FUNCTION_BLOCK CTRL_PI_AR (* AR-Adapter-Wrapper um OSCAT CTRL_PI - bruckt zwischen adapter und OSCAT PI-Regler. Istwert, Sollwert, Hand-Umschaltung, Handwert, Reglerparameter UND Rauschunterdrueckung/Offset/Grenzwerte vollstaendig als Adapter-Sockets - kein explizites REQ mehr noetig. *)
  (* Standard: 61499-2; Description: Copyright (c) 2026 Meisterschulen am Ostbahnhof This program and the accompanying materials are made available under the terms of the Eclipse Public License 2.0 which is available at https://www.eclipse.org/legal/epl-2.0/ SPDX-License-Identifier: EPL-2.0 *)
  (* Version 1.3, 2026-10-03, Franz Höpfinger, Meisterschulen am Ostbahnhof, Franz: 'auch umstellen auf Adapter Only' (analog CTRL_PID_AR v1.3/1.4) - SUP/OFS/LL/LH von InputVars (REAL, With-gebunden an REQ) auf AR-Adapter-Sockets umgestellt (gleiches Muster wie KP/KI/M_I: *.E1 loest CTRL_PI.REQ aus, *.D1 liefert den Wert). Explizites REQ-EventInput (inkl. With-Bindungen) und CNF-EventOutput komplett entfernt - CTRL_PI.CNF->E_D_FF_ANY.CLK bleibt intern bestehen (fuer das Latch von Y/DIFF/LIM), nur der externe CNF-Durchgriff entfaellt. RST unveraendert. Sockets/Connections/Dokumentation zugleich auf die Reihenfolge der CTRL_PI-InputVars sortiert: AR_ACT, SET, SUP, OFS, M_I, AX_MAN, KP, KI, LL, LH. *)
  (* Version 1.2, 2026-09-19, Franz Höpfinger, Meisterschulen am Ostbahnhof, Bugfix: REQ hatte keine With-Verknuepfung zu SUP/OFS/LL/LH (IEC 61499 - ungebundene Vars werden nicht zuverlaessig gelesen), jetzt ergaenzt, gespiegelt vom inneren CTRL_PI. M_I/KP/KI von InputVars auf AR-Adapter-Sockets umgestellt (Konsistenz mit AR_ACT/SET). *)
  (* Version 1.1, 2026-09-15, Franz Höpfinger, Meisterschulen am Ostbahnhof, INIT/INITO entfernt (CTRL_PI kennt kein INIT, nur REQ/RST) - stattdessen echtes REQ-EventInput/CNF-EventOutput ergaenzt, direkt auf CTRL_PI.REQ/CNF gemappt. SET von InputVar auf AR-Socket umgestellt (dynamisch berechneter Sollwert, wie AR_ACT) - SET.E1 triggert CTRL_PI.REQ zusaetzlich zu AR_ACT.E1/AX_MAN.E1. *)
  (* Version 1.0, 2026-09-12, Franz Höpfinger, Meisterschulen am Ostbahnhof, Initial implementation of CTRL_PI_AR wrapper FB *)
  PACKAGE OSCAT_adapter::Control;
  (* Documentation:
  CTRL_PI_AR
   🇩🇪 Deutsch
   AR-Adapter-Wrapper um OSCAT::Basic::POUs::Engineering::Control::CTRL_PI. Istwert (AR_ACT), Sollwert (SET), Rauschunterdrueckung/Offset (SUP/OFS), Handwert (M_I), Handbetrieb-Umschaltung (AX_MAN), Reglerparameter (KP/KI) UND Grenzwerte (LL/LH) sind als Adapter-Sockets ausgefuehrt, in derselben Reihenfolge wie die InputVars des umschlossenen CTRL_PI - jeder loest bei Ankunft eines neuen Werts CTRL_PI.REQ aus. Kein explizites REQ-Event mehr noetig, da jeder Socket selbst triggert. RST (Reset des Integrators) bleibt als eigenes Event erhalten.
   Reine Adapter-Grenze
    - AR_ACT (Socket, AR): Istwert (REAL, z. B. von FT_DERIV_10_AR.AR_OUT)
   - SET (Socket, AR): Sollwert (REAL, dynamisch berechnet, z. B. Fahrgeschwindigkeit*Voreilung)
   - SUP (Socket, AR): Rauschunterdrueckung (REAL, dynamisch)
   - OFS (Socket, AR): Offset (REAL, dynamisch)
   - M_I (Socket, AR): Handwert (REAL, dynamisch)
   - AX_MAN (Socket, AX): Handbetrieb-Umschaltung (optional, z. B. von AX_T_FF.Q)
   - KP/KI (Socket, AR): Reglerparameter (REAL, dynamisch)
   - LL/LH (Socket, AR): unterer/oberer Grenzwert (REAL, dynamisch)
   - AR_Y (Plug, AR): Stellwert (REAL, z. B. zur Weitergabe an AR_TO_AD_NUM.AR_IN)
   - AR_DIFF (Plug, AR): Regelabweichung (DIFF = SET - ACT, REAL)
   - AB_LIM (Plug, AB): Begrenzung aktiv Flag (LIM, BOOL)
    🇬🇧 English
   AR-adapter wrapper around OSCAT::Basic::POUs::Engineering::Control::CTRL_PI. Actual value (AR_ACT), set point (SET), noise suppression/offset (SUP/OFS), manual value (M_I), manual mode switch (AX_MAN), controller gains (KP/KI) AND limits (LL/LH) are all adapter sockets, in the same order as the wrapped CTRL_PI's own InputVars, each triggering CTRL_PI.REQ on arrival - no explicit REQ event needed any more, since every socket triggers itself. RST (integrator reset) remains its own event. Control output (AR_Y), control error (AR_DIFF) and limit flag (AB_LIM) are adapter plugs.
  *)
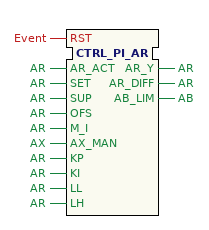
  EVENT_INPUT
    RST; (* Reset des Integrators (durchgereicht an CTRL_PI.RST) *)
  END_EVENT
  SOCKETS
    AR_ACT : adapter::types::unidirectional::AR; (* Istwert (REAL) *)
    SET : adapter::types::unidirectional::AR; (* Sollwert (REAL, dynamisch berechnet) *)
    SUP : adapter::types::unidirectional::AR; (* Rauschunterdrueckung (REAL, dynamisch) *)
    OFS : adapter::types::unidirectional::AR; (* Offset (REAL, dynamisch) *)
    M_I : adapter::types::unidirectional::AR; (* Handwert (REAL, dynamisch) *)
    AX_MAN : adapter::types::unidirectional::AX; (* Handbetrieb Umschaltung (BOOL/Event, optional) *)
    KP : adapter::types::unidirectional::AR; (* Proportionalbeiwert (REAL, dynamisch) *)
    KI : adapter::types::unidirectional::AR; (* Integralbeiwert (REAL, dynamisch) *)
    LL : adapter::types::unidirectional::AR; (* Unterer Grenzwert (REAL, dynamisch) *)
    LH : adapter::types::unidirectional::AR; (* Oberer Grenzwert (REAL, dynamisch) *)
  END_SOCKETS
  PLUGS
    AR_Y : adapter::types::unidirectional::AR; (* Stellwert (REAL) *)
    AR_DIFF : adapter::types::unidirectional::AR; (* Regelabweichung / Differenz (REAL) *)
    AB_LIM : adapter::types::unidirectional::AB; (* Begrenzung aktiv Flag (BOOL) *)
  END_PLUGS
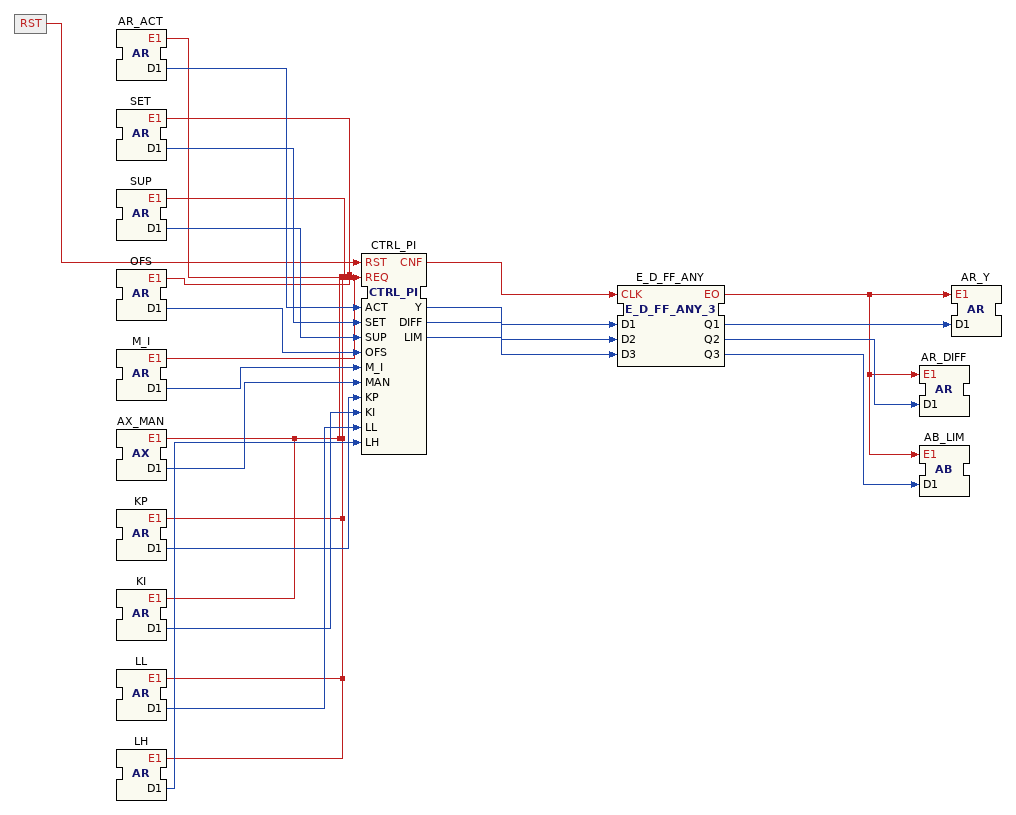
  FBS
    CTRL_PI : OSCAT::Basic::POUs::Engineering::Control::CTRL_PI;
    E_D_FF_ANY : iec61499::events::E_D_FF_ANY_3;
  END_FBS
  EVENT_CONNECTIONS
    RST TO CTRL_PI.RST;
    AR_ACT.E1 TO CTRL_PI.REQ;
    SET.E1 TO CTRL_PI.REQ;
    SUP.E1 TO CTRL_PI.REQ;
    OFS.E1 TO CTRL_PI.REQ;
    M_I.E1 TO CTRL_PI.REQ;
    AX_MAN.E1 TO CTRL_PI.REQ;
    KP.E1 TO CTRL_PI.REQ;
    KI.E1 TO CTRL_PI.REQ;
    LL.E1 TO CTRL_PI.REQ;
    LH.E1 TO CTRL_PI.REQ;
    CTRL_PI.CNF TO E_D_FF_ANY.CLK;
    E_D_FF_ANY.EO TO AR_Y.E1;
    E_D_FF_ANY.EO TO AR_DIFF.E1;
    E_D_FF_ANY.EO TO AB_LIM.E1;
  END_CONNECTIONS
  DATA_CONNECTIONS
    AR_ACT.D1 TO CTRL_PI.ACT;
    SET.D1 TO CTRL_PI.SET;
    SUP.D1 TO CTRL_PI.SUP;
    OFS.D1 TO CTRL_PI.OFS;
    M_I.D1 TO CTRL_PI.M_I;
    AX_MAN.D1 TO CTRL_PI.MAN;
    KP.D1 TO CTRL_PI.KP;
    KI.D1 TO CTRL_PI.KI;
    LL.D1 TO CTRL_PI.LL;
    LH.D1 TO CTRL_PI.LH;
    CTRL_PI.Y TO E_D_FF_ANY.D1;
    CTRL_PI.DIFF TO E_D_FF_ANY.D2;
    CTRL_PI.LIM TO E_D_FF_ANY.D3;
    E_D_FF_ANY.Q1 TO AR_Y.D1;
    E_D_FF_ANY.Q2 TO AR_DIFF.D1;
    E_D_FF_ANY.Q3 TO AB_LIM.D1;
  END_CONNECTIONS
END_FUNCTION_BLOCK
